// TIA Portal V17 export
// export: Created 2025-03-05T08:02:22.3723403Z, ExportSetting WithDefaults, DisplayName Totally Integrated Automation Portal, DisplayVersion V17 Update 8, DisplayName TIA Portal Openness, DisplayVersion V17 Update 8, DisplayName TIA Portal Version Control Interface, DisplayVersion V17, DisplayName SINAMICS Startdrive Advanced, DisplayVersion V17 SP2, DisplayName SINAMICS Startdrive G110M, G120, G120C, G120D, G120P, G115D, DisplayVersion V17 SP2, DisplayName SINAMICS Startdrive G130, G150, S120, S150, SINAMICS MV, S210, DisplayVersion V17 SP2, DisplayName STEP 7 Professional, DisplayVersion V17 Update 8, DisplayName SINUMERIK ONE STEP 7 Toolbox, DisplayVersion V17 Update 12, DisplayName SINUMERIK 840D sl STEP 7 Toolbox, DisplayVersion V17 Update 12, DisplayName STEP 7 Safety, DisplayVersion V17 Update 6, DisplayName WinCC Advanced, DisplayVersion V17 Update 8
TYPE "MR_J4_TN_Output"
// stored: IsFailsafeCompliant false
   STRUCT
      Output : Struct
         "Q_Mode opeation_B1" : Byte;
         "Q_Mode opeation_B2" : Byte;
         Q_CW_B8_Halt : Bool;
         Q_CW_B9_ChangeP2 : Bool;
         Q_CW_B10 : Bool;
         Q_CW_B11 : Bool;
         Q_CW_B12 : Bool;
         Q_CW_B13 : Bool;
         Q_CW_B14 : Bool;
         Q_CW_B15 : Bool;
         Q_CW_B0_SO : Bool;
         Q_CW_B1_EV : Bool;
         Q_CW_B2_QS : Bool;
         Q_CW_B3_EO : Bool;
         Q_CW_B4_Npoint : Bool;
         Q_CW_B5_ChangeP : Bool;
         Q_CW_B6_Abs_Rel : Bool;
         Q_CW_B7_FReset : Bool;
         "Q_Control DI 1" : Word;
         "Q_Control D12" : Word;
         "Q_Control DI 3" : Word;
         "Q_Target torque" : Int;
         "Q_Torque Slope" : DInt;
         "Q_Target position" : DInt;
         "Q_Taget velocity" : DInt;
         "Q_Velocity limit" : DInt;
         "Q_Profile velocity" : DInt;
         "Q_Profile acceleration" : DInt;
         "Q_Profile deeleration" : DInt;
         "Q_Touch probe" : Word;
         Q_reserved1 : Word;
         Q_reserved2 : Word;
         Q_reserved3 : Word;
      END_STRUCT;
   END_STRUCT;
END_TYPE
